(*
used to create event schedulers
*)

FUNCTION_BLOCK ABSTRACT FB_EventScheduler
VAR_INPUT
END_VAR
VAR_OUTPUT
END_VAR
VAR
END_VAR

gh

END_FUNCTION_BLOCK

(* stored: Version 1.1.0.1, ProductVersion 3.1.4024.12
   POU FB_EventScheduler: Id {b24ddb6a-18e7-4e58-a78a-64df0d31999b}, SpecialFunc None *)
